// TIA Portal project "AWL EJEMPLOS" (V11)

(* hardware
DEVICE "S7300/ET200 station_1"  SIMATIC 300-Station
   slot 0: "Perfil soporte_0"  Rail  6ES7 390-1***0-0AA0
   slot 2: "PLC_1"  CPU 313C-2 DP  6ES7 313-6CF03-0AB0  V2.6
      slot 0: "Interfaz MPI_1"  MPI
      slot 1: "Interfaz DP_1"  DP
      slot 2: "DI16/DO16_1"  DI16/DO16
      slot 4: "Contaje_1"  Counter
*)

// ===== PLC "PLC_1"  CPU 313C-2 DP =====

VAR_GLOBAL   // PLC tag table "Tabla de variables estándar"
   "Tag_1" AT %E0.0 : Bool;
   "Tag_2" AT %E0.1 : Bool;
   "Tag_3" AT %A0.0 : Bool;
   "Tag_4" AT %A0.1 : Bool;
   "Tag_5" AT %A0.2 : Bool;
   "Tag_6" AT %E0.2 : Bool;
   "Tag_7" AT %E0.3 : Bool;
   "Tag_8" AT %E0.4 : Bool;
   "Tag_9" AT %M0.0 : Bool;
   "Tag_10" AT %E0.5 : Bool;
   "Tag_11" AT %A0.4 : Bool;
   "Tag_12" AT %A0.3 : Bool;
END_VAR

DATA_BLOCK "Bloque_1_DB"   // DB1
{ S7_Optimized_Access := 'FALSE' }
VERSION : 0.1
// stored: InstanceOfName 3 L ENCENDIDO CONDICIONAL
"3 L  ENCENDIDO CONDICIONAL"
BEGIN
END_DATA_BLOCK

DATA_BLOCK "3 L  ENCENDIDO CONDICIONAL_DB"   // DB2
{ S7_Optimized_Access := 'FALSE' }
VERSION : 0.1
// stored: InstanceOfName 3 L ENCENDIDO CONDICIONAL
"3 L  ENCENDIDO CONDICIONAL"
BEGIN
END_DATA_BLOCK

DATA_BLOCK "FLANCOS"   // DB3
{ S7_Optimized_Access := 'FALSE' }
VERSION : 0.1
   VAR
      F0 : Bool;
      F1 : Bool;
      F2 : Bool;
      F3 : Bool;
      F4 : Bool;
      F5 : Bool;
      F6 : Bool;
      F7 : Bool;
      B0 : Bool;
      B1 : Bool;
      B2 : Bool;
      B3 : Bool;
      B4 : Bool;
      B5 : Bool;
      B6 : Bool;
      B7 : Bool;
   END_VAR
BEGIN
END_DATA_BLOCK

DATA_BLOCK "MARCHA /PARO 1 P_DB"   // DB4
{ S7_Optimized_Access := 'FALSE' }
VERSION : 0.1
// stored: InstanceOfName MARCHA /PARO 1 P
"MARCHA /PARO 1 P"
BEGIN
END_DATA_BLOCK

FUNCTION_BLOCK "3 L  ENCENDIDO CONDICIONAL"   // FB1, STL
{ S7_Optimized_Access := 'FALSE' }
VERSION : 0.1
   VAR_INPUT
      "PARO 1" : Bool;
      "PARO 2" : Bool;
      "MARCHA 1" : Bool;
      "MARCHA 2" : Bool;
      "MARCHA 3" : Bool;
   END_VAR
   VAR_OUTPUT
      L1 : Bool;
      L2 : Bool;
      L3 : Bool;
   END_VAR
BEGIN

REGION Network 1
         O     #"PARO 1";  //PARO 1
         O     #"PARO 2";  //PARO 2
         R     #L1;
         R     #L2;
         R     #L3;
         ON    #L2;
         O     #L3;
         A     #"MARCHA 1";  //MARCHA 1
         S     #L1;  //LAMPARA 1
         ON    #L1;
         O     #L3;
         A     #"MARCHA 2";  //MARCHA 2
         S     #L2;  //LAMPARA 2
         A     #"MARCHA 3";  //MARCHA 3
         S     #L3;  //LAMPARA 3
END_REGION
END_FUNCTION_BLOCK

FUNCTION_BLOCK "MARCHA /PARO 1 P"   // FB2, STL
{ S7_Optimized_Access := 'FALSE' }
VERSION : 0.1
   VAR_INPUT
      "MARCHA/PARO" : Bool;
   END_VAR
   VAR_OUTPUT
      "LAMPARA 1" : Bool;
   END_VAR
BEGIN

REGION Network 1
         A     #"MARCHA/PARO";  //P
         FP    "FLANCOS".F0;
         AN    #"LAMPARA 1";
         =     "FLANCOS".B0;  // PULASO 1
         A     #"MARCHA/PARO";  // P
         FP    "FLANCOS".F1;
         A     #"LAMPARA 1";
         =     "FLANCOS".B1;  // PULSO 2
         A     "FLANCOS".B0;
         S     #"LAMPARA 1";
         A     "FLANCOS".B1;
         R     #"LAMPARA 1";
END_REGION
END_FUNCTION_BLOCK

ORGANIZATION_BLOCK "Main"   // OB1, LAD
TITLE = "Main Program Sweep (Cycle)"
{ S7_Optimized_Access := 'FALSE' }
VERSION : 0.1
   VAR_TEMP
      OB1_EV_CLASS : Byte;   // Bits 0-3 = 1 (Coming event), Bits 4-7 = 1 (Event class 1)
      OB1_SCAN_1 : Byte;   // 1 (Cold restart scan 1 of OB 1), 3 (Scan 2-n of OB 1)
      OB1_PRIORITY : Byte;   // Priority of OB Execution
      OB1_OB_NUMBR : Byte;   // 1 (Organization block 1, OB1)
      OB1_RESERVED_1 : Byte;   // Reserved for system
      OB1_RESERVED_2 : Byte;   // Reserved for system
      OB1_PREV_CYCLE : Int;   // Cycle time of previous OB1 scan (milliseconds)
      OB1_MIN_CYCLE : Int;   // Minimum cycle time of OB1 (milliseconds)
      OB1_MAX_CYCLE : Int;   // Maximum cycle time of OB1 (milliseconds)
      OB1_DATE_TIME : Date_And_Time;   // Date and time OB1 started
   END_VAR
BEGIN

REGION Network 1
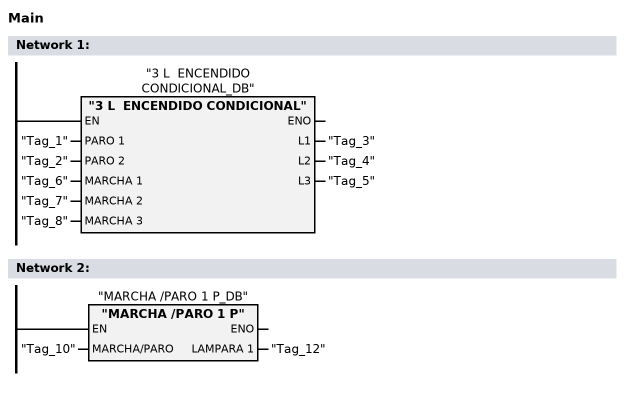
   RUNG wire#powerrail
      "3 L  ENCENDIDO CONDICIONAL_DB"("PARO 1" := "Tag_1", "PARO 2" := "Tag_2", "MARCHA 1" := "Tag_6", "MARCHA 2" := "Tag_7", "MARCHA 3" := "Tag_8", L1 => "Tag_3", L2 => "Tag_4", L3 => "Tag_5")
   END_RUNG
   // the same network as SCL:
   "3 L  ENCENDIDO CONDICIONAL_DB"("PARO 1" := "Tag_1",   // "3 L  ENCENDIDO CONDICIONAL"
                           "PARO 2" := "Tag_2",
                           "MARCHA 1" := "Tag_6",
                           "MARCHA 2" := "Tag_7",
                           "MARCHA 3" := "Tag_8",
                           L1 => "Tag_3",
                           L2 => "Tag_4",
                           L3 => "Tag_5");
END_REGION

REGION Network 2
   RUNG wire#powerrail
      "MARCHA /PARO 1 P_DB"("MARCHA/PARO" := "Tag_10", "LAMPARA 1" => "Tag_12")
   END_RUNG
   // the same network as SCL:
   "MARCHA /PARO 1 P_DB"("MARCHA/PARO" := "Tag_10", "LAMPARA 1" => "Tag_12");   // "MARCHA /PARO 1 P"
END_REGION
END_ORGANIZATION_BLOCK